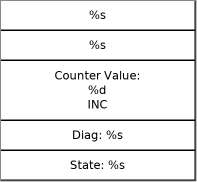
VISUALIZATION TplTsConnectionEL5021  // 197x182
VAR_IN_OUT
	stConnectionDiag 			:FB_TwinSafeConnectionEL5021;
END_VAR
(* End *)
    Rectangle (0,0 195x30), "%s", text variable: stConnectionDiag.sEcSlaveName, colour toggle: stConnectionDiag.sDiag = 'No error'
    Rectangle (0,60 195x60), "Counter Value: %d INC", text variable: stConnectionDiag.nInSafeDataCounterValue
    Rectangle (0,120 195x30), "Diag: %s", text variable: stConnectionDiag.sDiag, colour toggle: stConnectionDiag.sDiag <> 'No error'
    Rectangle (0,150 195x30), "State: %s", text variable: stConnectionDiag.sState
    Rectangle (0,30 195x30), "%s", text variable: stConnectionDiag.sEcSlaveType
END_VISUALIZATION

(* stored: Version 1.1.0.1
   Visu TplTsConnectionEL5021: Id {3424a977-91f9-449a-bc2a-bb85843d3caa} *)
